// TwinCAT 3 PLC project HOMS_XRT_PLC
// Title: lcls-plc-xrt-optics
// Company: SLAC
// ProjectVersion: 4.4.0
// ProgramVersion: 3.1.4022.7
// CompilerDefines: L
// libraries:
//   lcls-twincat-motion, * (SLAC)
//   lcls-twincat-optics, * (SLAC)
//   PMPS, * (SLAC - LCLS)
//   Tc2_ControllerToolbox, * (Beckhoff Automation GmbH)
//   Tc2_EtherCAT, * (Beckhoff Automation GmbH)
//   Tc2_MC2, * (Beckhoff Automation GmbH)
//   Tc2_SerialCom, * (Beckhoff Automation GmbH)
//   Tc2_Standard, * (Beckhoff Automation GmbH)
//   Tc2_System, * (Beckhoff Automation GmbH)
//   Tc2_Utilities, * (Beckhoff Automation GmbH)
//   Tc3_Module, * (Beckhoff Automation GmbH)
//   VisuDialogs, * (System)
//   LCLS General,2.4.2,SLAC
// project tree:
//   Common/DUTs/ ENUM_Coating_States.TcDUT (not stored), E_GantryControl.TcDUT (not stored), E_GantryMode.TcDUT (not stored), E_PiezoControl.TcDUT (not stored), E_PitchControl.TcDUT (not stored), HOMS_Gantry.TcDUT (not stored), HOMS_GantryAxis.TcDUT (not stored), HOMS_PitchMechanismOld.TcDUT (not stored), ST_AbstractAxis.TcDUT (not stored), ST_CoEIndSub.TcDUT (not stored), ST_DecoupledMotionPermits.TcDUT (not stored), ST_ElmoGDCBellCoEParams.TcDUT (not stored), ST_HOMSStepper.TcDUT (not stored), ST_PiezoAxisOld.TcDUT (not stored), ST_StepperStatus.TcDUT (not stored)
//   Version/ Global_Version.TcGVL
//   Common/POUs/Helpers/ FB_Drive.TcPOU (not stored), FB_ElmoGDCBellCoE.TcPOU (not stored), FB_ElmoMCUploadDriveParams.TcPOU (not stored), FB_ElmoStoMonitor.TcPOU (not stored), FB_GantryDiffVirtualLimitSwitch.TcPOU (not stored), FB_InitDriveRefs.TcPOU (not stored), FB_LimitSwitchState.TcPOU (not stored), FB_PitchSoftLimits.TcPOU (not stored), FB_PI_E621_SerialDriverOld.TcPOU (not stored), FB_PI_E621_SerialTransaction.TcPOU (not stored), FB_PTP.TcPOU (not stored), FB_ReadFloatParameter.TcPOU (not stored), FB_ReadParameterInNC.TcPOU (not stored), FB_WriteParameterInNC.TcPOU (not stored), F_PiezoPosition.TcPOU (not stored), MC_SmoothMover.TcPOU (not stored), WithinRange.TcPOU (not stored)
//   Common/POUs/HOMS_FBs/ FB_Gantry.TcPOU (not stored), FB_GantryDifferenceMonitor.TcPOU (not stored), FB_PiezoControl.TcPOU (not stored), FB_PitchControlOld.TcPOU (not stored), FB_ReduceGantryDiff.TcPOU (not stored)
//   / GlobalTextList.TcGTLO (not stored), PiezoDriver.TcTTO (not stored), PlcTask.TcTTO (not stored), SerialIO.TcTTO (not stored), Visualization Manager.TcVMO (not stored)
//   GVLs/ GVL.TcGVL (not stored), GVL_COM_Buffers.TcGVL (not stored), GVL_Constants.TcGVL (not stored), GVL_MR1L3.TcGVL (not stored), GVL_MR1L4_Constants.TcGVL (not stored), GVL_MR1L4.TcGVL (not stored), GVL_MR1L3_Constants.TcGVL (not stored), GVL_MR2L3_Constants.TcGVL (not stored), GVL_MR2L3.TcGVL (not stored), GVL_PMPS.TcGVL (not stored), GVL_RTDS.TcGVL (not stored), GVL_SerialIO.TcGVL (not stored)
//   POUs/ FB_Coating_States_noPMPS.TcPOU (not stored), FB_MirrorCoatingProtection.TcPOU (not stored), FB_Coating_States.TcPOU (not stored), Main.TcPOU (not stored), PRG_PMPS.TcPOU (not stored), PRG_CoatingProtection.TcPOU (not stored)
//   POUs/Serial Comm/ PiezoSerial.TcPOU (not stored), P_Serial_Com.TcPOU (not stored)
//   VISUs/ GantryControls.TcVIS (not stored), Visualization.TcVIS (not stored), PiezoControls.TcVIS (not stored)

// ---- Version/Global_Version.TcGVL
{attribute 'TcGenerated'}
// This function has been automatically generated from the project information.
VAR_GLOBAL CONSTANT
    {attribute 'const_non_replaced'}
    {attribute 'linkalways'}
    stLibVersion_lcls_plc_xrt_optics : ST_LibVersion := (iMajor := 4, iMinor := 4, iBuild := 0, iRevision := 0, sVersion := '4.4.0');
END_VAR
